Staubli VAL3: flushQueue.pgx

public program flushQueue(num x_nConvNum (dimensions=1), num& x_nError[] (dimensions=1))
begin
  // This program flushes the queue of objects.
  //
  // Input Param
  //  x_nConvNum : Conveyor number
  //
  // Output param
  //  x_nError    : Error code
  //    0    --> No error
  //    3    --> Invalid conveyor number
  //
  //----------------------------------------------------------------
  //
  x_nError=0
  switch x_nConvNum
    case 0
      call cnv0:flushQueue()
    break
    case 1
      call cnv1:flushQueue()
    break
    default
      x_nError=3
    break
  endSwitch
end
